GLOBALCONSTANTS AID_CO (* Container object attribute ids (all read-only) *)
  (* Standard: 61499-1; Description: Copyright (c) 2023 HR Agrartechnik GmbH This program and the accompanying materials are made available under the terms of the Eclipse Public License 2.0 which is available at https://www.eclipse.org/legal/epl-2.0/ SPDX-License-Identifier: EPL-2.0 *)
  (* Version 1.0, 2026-06-20, Franz Höpfinger, HR Agrartechnik GmbH *)
  PACKAGE isobus::UT::Q::const::AID;
  VAR_GLOBAL CONSTANT
    WIDTH : USINT := USINT#1; (* 1: AID_CO_WIDTH - [1] Read-only for Change Attribute (ISO 11783-6). Query via Get Attribute Value (F.58). Maximum width of the container's area in pixels. *)
    HEIGHT : USINT := USINT#2; (* 2: AID_CO_HEIGHT - [2] Read-only for Change Attribute (ISO 11783-6). Query via Get Attribute Value (F.58). Maximum height of the container's area in pixels. *)
    HIDDEN : USINT := USINT#3; (* 3: AID_CO_HIDDEN - [3] Read-only for Change Attribute (ISO 11783-6). Query via Get Attribute Value (F.58); manage via Hide/Show Object (F.2). *)
  END_VAR
END_GLOBALCONSTANTS
